TYPE WcStateInputToggleBase_F68C23A9 :
STRUCT
END_STRUCT
END_TYPE

(* stored: Version 1.2.0.0, ProductVersion 3.1.4024.9
   DUT WcStateInputToggleBase_F68C23A9: Id {448080d7-799a-4cae-a336-1daa4a7832c1} *)
